// TIA Portal V19 export
FUNCTION "FC903_SafetyOutputs" : Void   // FC903, F_LAD
{ S7_Optimized_Access := 'TRUE' }
// stored: AutoNumber false
   VAR CONSTANT
      ct_FeedbackTime : Time := T#300ms;
   END_VAR
BEGIN

REGION Network 1: Enable air pressure supply on the left robot
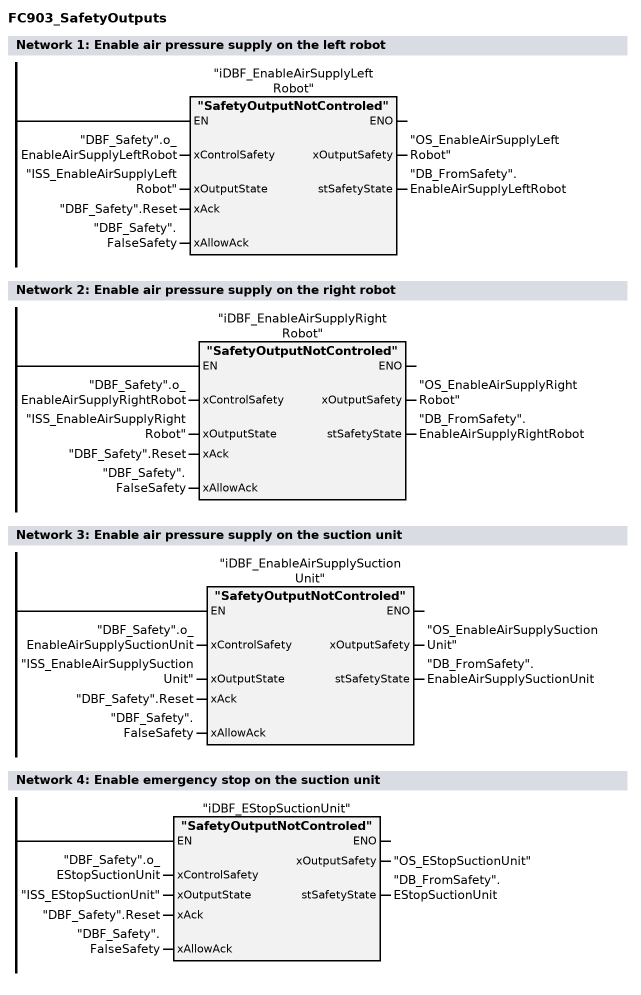
   RUNG wire#powerrail
      "iDBF_EnableAirSupplyLeftRobot"(xControlSafety := "DBF_Safety".o_EnableAirSupplyLeftRobot, xOutputState := "ISS_EnableAirSupplyLeftRobot", xAck := "DBF_Safety".Reset, xAllowAck := "DBF_Safety".FalseSafety, xOutputSafety => "OS_EnableAirSupplyLeftRobot", stSafetyState => "DB_FromSafety".EnableAirSupplyLeftRobot)
   END_RUNG
   // the same network as SCL:
   "iDBF_EnableAirSupplyLeftRobot"(xControlSafety := "DBF_Safety".o_EnableAirSupplyLeftRobot,   // "SafetyOutputNotControled"
                           xOutputState := "ISS_EnableAirSupplyLeftRobot",
                           xAck := "DBF_Safety".Reset,
                           xAllowAck := "DBF_Safety".FalseSafety,
                           xOutputSafety => "OS_EnableAirSupplyLeftRobot",
                           stSafetyState => "DB_FromSafety".EnableAirSupplyLeftRobot);
END_REGION

REGION Network 2: Enable air pressure supply on the right robot
   RUNG wire#powerrail
      "iDBF_EnableAirSupplyRightRobot"(xControlSafety := "DBF_Safety".o_EnableAirSupplyRightRobot, xOutputState := "ISS_EnableAirSupplyRightRobot", xAck := "DBF_Safety".Reset, xAllowAck := "DBF_Safety".FalseSafety, xOutputSafety => "OS_EnableAirSupplyRightRobot", stSafetyState => "DB_FromSafety".EnableAirSupplyRightRobot)
   END_RUNG
   // the same network as SCL:
   "iDBF_EnableAirSupplyRightRobot"(xControlSafety := "DBF_Safety".o_EnableAirSupplyRightRobot,   // "SafetyOutputNotControled"
                           xOutputState := "ISS_EnableAirSupplyRightRobot",
                           xAck := "DBF_Safety".Reset,
                           xAllowAck := "DBF_Safety".FalseSafety,
                           xOutputSafety => "OS_EnableAirSupplyRightRobot",
                           stSafetyState => "DB_FromSafety".EnableAirSupplyRightRobot);
END_REGION

REGION Network 3: Enable air pressure supply on the suction unit
   RUNG wire#powerrail
      "iDBF_EnableAirSupplySuctionUnit"(xControlSafety := "DBF_Safety".o_EnableAirSupplySuctionUnit, xOutputState := "ISS_EnableAirSupplySuctionUnit", xAck := "DBF_Safety".Reset, xAllowAck := "DBF_Safety".FalseSafety, xOutputSafety => "OS_EnableAirSupplySuctionUnit", stSafetyState => "DB_FromSafety".EnableAirSupplySuctionUnit)
   END_RUNG
   // the same network as SCL:
   "iDBF_EnableAirSupplySuctionUnit"(xControlSafety := "DBF_Safety".o_EnableAirSupplySuctionUnit,   // "SafetyOutputNotControled"
                           xOutputState := "ISS_EnableAirSupplySuctionUnit",
                           xAck := "DBF_Safety".Reset,
                           xAllowAck := "DBF_Safety".FalseSafety,
                           xOutputSafety => "OS_EnableAirSupplySuctionUnit",
                           stSafetyState => "DB_FromSafety".EnableAirSupplySuctionUnit);
END_REGION

REGION Network 4: Enable emergency stop on the suction unit
   RUNG wire#powerrail
      "iDBF_EStopSuctionUnit"(xControlSafety := "DBF_Safety".o_EStopSuctionUnit, xOutputState := "ISS_EStopSuctionUnit", xAck := "DBF_Safety".Reset, xAllowAck := "DBF_Safety".FalseSafety, xOutputSafety => "OS_EStopSuctionUnit", stSafetyState => "DB_FromSafety".EStopSuctionUnit)
   END_RUNG
   // the same network as SCL:
   "iDBF_EStopSuctionUnit"(xControlSafety := "DBF_Safety".o_EStopSuctionUnit,   // "SafetyOutputNotControled"
                           xOutputState := "ISS_EStopSuctionUnit",
                           xAck := "DBF_Safety".Reset,
                           xAllowAck := "DBF_Safety".FalseSafety,
                           xOutputSafety => "OS_EStopSuctionUnit",
                           stSafetyState => "DB_FromSafety".EStopSuctionUnit);
END_REGION
END_FUNCTION
